// TIA Portal V20 export
// export: Created 2026-10-03T18:54:34.4362638Z, ExportSetting WithDefaults, DisplayName Totally Integrated Automation Portal, DisplayVersion V20 Update 4, DisplayName TIA Portal Openness, DisplayVersion V20 Update 4, DisplayName TIA Portal Version Control Interface, DisplayVersion V20 Update 4, DisplayName SINAMICS Startdrive Advanced, DisplayVersion V20 SP1 Update 1, DisplayName SINAMICS Startdrive G110M, G120, G120C, G120D, G120P, G115D, DisplayVersion V20 SP1 Update 1, DisplayName SINAMICS Startdrive G130, G150, S120, S150, SINAMICS MV, G220, S200, S210, DisplayVersion V20 SP1 Update 1, DisplayName STEP 7 Professional, DisplayVersion V20 Update 4, DisplayName STEP 7 Safety, DisplayVersion V20 Update 2, DisplayName WinCC Basic/Comfort/Advanced, DisplayVersion V20 Update 4, DisplayName WinCC Unified, DisplayVersion V20 Update 4
FUNCTION "SLC_FLOAT_READ" : Real   // FC16, SCL
TITLE = Read a float by file and element number
{ S7_Optimized_Access := 'TRUE' }
VERSION : 0.1
// Reads F<File>:<Element> where the element (or file) number comes from another word, as in the SLC indirect
//  address F90:[N7:55].
// stored: AutoNumber true, IsIECCheckEnabled false, SetENOAutomatically false, UDAEnableTagReadback false
   VAR_INPUT
      File : DInt;   // Float file number (90 for F90)
      Element : DInt;   // Element number
   END_VAR
BEGIN
   // 16#84 is the DB memory area; each float is 4 bytes.
   #SLC_FLOAT_READ := DWORD_TO_REAL(PEEK_DWORD(area := 16#84, dbNumber := #File, byteOffset := #Element * 4));
END_FUNCTION
